// SIMATIC S7-200 project (STEP 7-Micro/WIN), CPU 221 REL 01.10

SYMBOL_TABLE USER1
start            I0.0
estop            I0.1
DC               Q0.0
END_SYMBOL_TABLE

ORGANIZATION_BLOCK MAIN:OB1
TITLE=PROGRAM COMMENTS
BEGIN
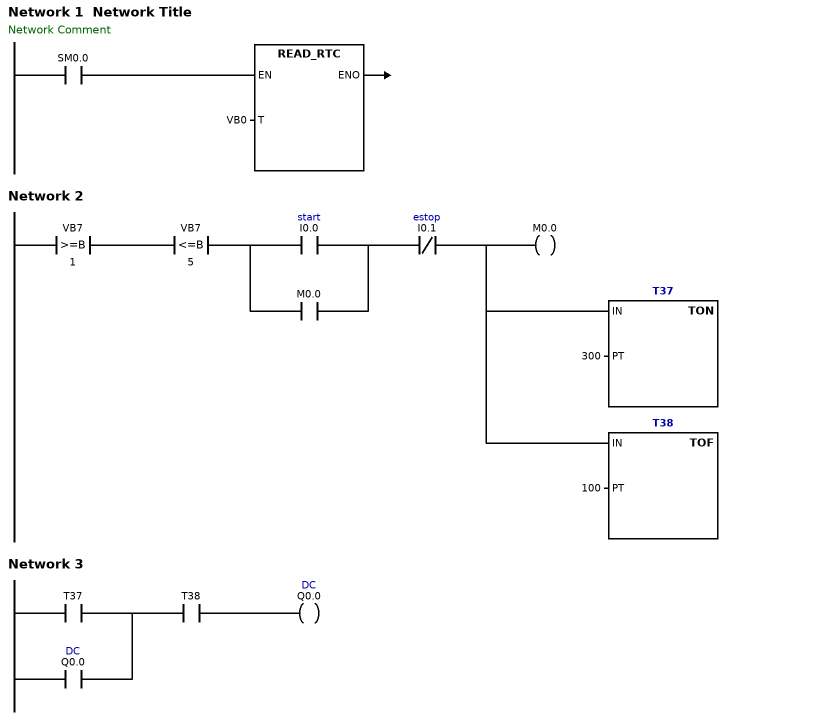
Network 1 // Network Title
// Network Comment
LD     SM0.0
TODR   VB0
Network 2
LDB>=  VB7, 1
AB<=   VB7, 5
LD     start:I0.0
O      M0.0
ALD
AN     estop:I0.1
=      M0.0
TON    T37, 300
TOF    T38, 100
Network 3
LD     T37
O      DC:Q0.0
A      T38
=      DC:Q0.0
END_ORGANIZATION_BLOCK
